(*
    This test-suite runs several asserts with the same parameters (same expected, actual, message) in the same cycle.
    The reason we want the framework to support this is that theoretically the user could want to do an assert with the
    same message, in the same test, with the same data values for both expected and actual, although the data that the
    user does the assert on might be from different data sets.
*)
{attribute 'call_after_init'}
FUNCTION_BLOCK FB_MultipleAssertWithSameParametersInSameCycle EXTENDS TcUnit.FB_TestSuite IMPLEMENTS TcUnit.I_RunnableTestSuite
VAR
    Assert : TcUnit.FB_Assert;
END_VAR

METHOD PRIVATE Assert_SeveralTimes
VAR
    a : DWORD := 16#12345678;
    b : DWORD := 16#90ABCDEF;
END_VAR
TEST('Assert_SeveralTimes');

Assert.AssertEquals_DWORD(Expected := a,
                          Actual := b,
                          Message := 'Values differ');

Assert.AssertEquals_DWORD(Expected := a,
                          Actual := b,
                          Message := 'Values differ');
END_METHOD

METHOD FB_init : BOOL
VAR_INPUT
	bInitRetains : BOOL; // if TRUE, the retain variables are initialized (warm start / cold start)
	bInCopyCode : BOOL;  // if TRUE, the instance afterwards gets moved into the copy code (online change)
END_VAR
SUPER^.RegisterTestSuite(THIS^);
END_METHOD

METHOD PUBLIC RunTests : TCUNIT.E_TestSuiteRunState
Assert_SeveralTimes();

RunTests := TCUNIT.E_TestSuiteRunState.FINISHED;
END_METHOD

END_FUNCTION_BLOCK

(* stored: Version 1.1.0.1, ProductVersion 3.1.4022.16
   POU FB_MultipleAssertWithSameParametersInSameCycle: Id {9957a11f-d554-4b5d-be35-f56d53aab4f2}, SpecialFunc None
   Method Assert_SeveralTimes: Id {cd07d59b-c5ef-4bab-a334-9a8ba622ccca}
   Method FB_init: Id {efb41198-520b-42d0-bc0b-dbcbcf350121}
   Method RunTests: Id {77cf1a7c-08aa-49c0-bcbe-1902ef9f2ce2} *)
